Staubli VAL3: Move.pgx

program Move(num& arrayValue[])
  local pointRx pt
begin
//*******************************************************************************
//*   ______
//*  / _____) /|
//* | |      / /
//* | | /\  / /
//* | | \ \/ /  _      Copyright (c) KEOLABS, 2016
//* | |  \__/  | |        http://www.keolabs.com
//* | |________| |
//*  \__________/
//*
//********************************************************************************
//*@file          : Move
//*@author        : Yves Ragot
//*@version       : $Id: Move.pgx 1198 2016-10-07 06:48:14Z yves $
//*@brief         : Move command treatment (relative mouvement)
//*
//*******************************************************************************/

  // current Cartesian position
  pt = here(tCurrentTool, fCurrentFrame)

  // get and compute target point
  pTargetPoint.trsf.x = pt.trsf.x + arrayValue[0]
  pTargetPoint.trsf.y = pt.trsf.y + arrayValue[1]
  pTargetPoint.trsf.z = pt.trsf.z + arrayValue[2]
  pTargetPoint.trsf.rx = pt.trsf.rx + arrayValue[3]
  pTargetPoint.trsf.ry = pt.trsf.ry + arrayValue[4]
  pTargetPoint.trsf.rz = pt.trsf.rz + arrayValue[5]

  CartesianMode = true

  // launch mouvement
  ExecuteMotion = true

  // wait for end of execution
  wait(ExecuteMotion == false)

end
